(*
SPDX-FileCopyrightText: © 2026 Oleksandr Tiutyk <trofimich@gmail.com>
SPDX-License-Identifier: MIT
License: https://opensource.org/license/mit
*)

FUNCTION_BLOCK StringHelperTest EXTENDS TcUnit.FB_TestSuite
VAR
	{attribute 'hide'} 
	_ClassName : STRING := __POUNAME();
END_VAR

AppendToTarget();
ReplaceInSource();
Split();
Join();
Trim();

METHOD AppendToTarget
VAR
	testString : STRING;

	expectedString : STRING := 'Original string + first appended string + second appended string';
	
	stringToAppend_1 : STRING := 'first appended string';
	stringToAppend_2 : STRING := 'second appended string';
	plusString : STRING := ' + ';
	
	result : BOOL;
END_VAR
VAR_INST
	testFinished : BOOL;
END_VAR
IF testFinished THEN 
	RETURN; 
END_IF 

TEST(__POUNAME());

testString := 'Original string';
TOF_Core.Strings.AppendToTarget255(testString, ' + ', stringToAppend_1, ' + ', stringToAppend_2);
AssertEquals_STRING(expectedString, testString, 'Invalid String.AppendToTarget255 method result');

testString := 'Original string';
result := TOF_Core.Strings.TryAppendToTarget255(testString, ' + ', stringToAppend_1, ' + ', stringToAppend_2);
AssertEquals_STRING(expectedString, testString, 'Invalid String.TryAppendToTarget255 method result');
AssertEquals_BOOL(result, TRUE, 'Invalid String.TryAppendToTarget255 method returned result');

result := TOF_Core.Strings.TryAppendToTarget255(testString, ' + ', stringToAppend_1);
AssertEquals_BOOL(result, FALSE, 'Invalid String.TryAppendToTarget255 method returned result');

testString := 'Original string';
TOF_Core.Strings.AppendToTarget(testString, plusString);
TOF_Core.Strings.AppendToTarget(testString, stringToAppend_1);
TOF_Core.Strings.AppendToTarget(testString, plusString);
TOF_Core.Strings.AppendToTarget(testString, stringToAppend_2);
AssertEquals_STRING(expectedString, testString, 'Invalid String.AppendToTarget method result');

testString := 'Original string';
result := TOF_Core.Strings.TryAppendToTarget(testString, plusString)
	AND TOF_Core.Strings.TryAppendToTarget(testString, stringToAppend_1)
	AND TOF_Core.Strings.TryAppendToTarget(testString, plusString)
	AND TOF_Core.Strings.TryAppendToTarget(testString, stringToAppend_2);
AssertEquals_STRING(expectedString, testString, 'Invalid String.TryAppendToTarget method result');
AssertEquals_BOOL(result, TRUE, 'Invalid String.TryAppendToTarget method returned result');

result := TOF_Core.Strings.TryAppendToTarget(testString, plusString)
	AND TOF_Core.Strings.TryAppendToTarget(testString, stringToAppend_1);
AssertEquals_BOOL(result, FALSE, 'Invalid String.TryAppendToTarget method returned result');

testFinished := TRUE; 
TEST_FINISHED();
END_METHOD

{attribute 'monitoring' := 'call'}
PROPERTY ClassName : REFERENCE TO STRING
GET
ClassName REF= _ClassName;
END_GET
END_PROPERTY

METHOD Join
VAR
	stringToSplit : STRING := '123 , , 456, 789 ,0';
	separator : STRING := ',';
	
	splitter : TOF_Core.StringSplittingEnumerator;

	joinedString1, joinedString2 : STRING;
END_VAR
VAR_INST
	testFinished : BOOL;
END_VAR
IF testFinished THEN 
	RETURN; 
END_IF 

TEST(__POUNAME());

// simple splitting
splitter := TOF_Core.Strings.CreateSplitter(stringToSplit, separator);

// simple joining
TOF_Core.Strings.JoinToTarget(joinedString1, separator, splitter);

AssertEquals_STRING(stringToSplit, joinedString1, TOF_Core.Strings.Concat255('Invalid first Strings.JoinToTarget result string ', joinedString1));

// splitting with maxCount, trimming and empty string removing 
splitter := TOF_Core.Strings.CreateSplitter(stringToSplit, separator, 3, TRUE, TRUE);

// joining with startIndex and count
TOF_Core.Strings.JoinToTarget(joinedString2, separator, splitter, 1, 2);

AssertEquals_STRING('456,789', joinedString2, TOF_Core.Strings.Concat255('Invalid second Strings.JoinToTarget result string ', joinedString2));

testFinished := TRUE;
TEST_FINISHED();
END_METHOD

{attribute 'monitoring' := 'call'}
PROPERTY NamespaceName : REFERENCE TO STRING
GET
NamespaceName REF= CurrentNamespace.Name;
END_GET
END_PROPERTY

METHOD ReplaceInSource
VAR
	testString : STRING(18);
	
	replacementCount : UINT;
	result : BOOL;
END_VAR
VAR_INST
	testFinished : BOOL;
END_VAR
IF testFinished THEN 
	RETURN; 
END_IF 

TEST(__POUNAME());

testString := 'abcd_abcd_abcd';
TOF_Core.Strings.ReplaceInSource(testString, 'bc', '0', replacementCount => replacementCount);
AssertEquals_STRING('a0d_a0d_a0d', testString, 'Invalid String.ReplaceInSource result string');
AssertEquals_UINT(3, replacementCount, 'Invalid String.ReplaceInSource replacingCount count');

testString := 'abcd_abcd_abcd';
TOF_Core.Strings.ReplaceInSource(testString, 'bc', '123', replacementCount => replacementCount);
AssertEquals_STRING('a123d_a123d_a123d', testString, 'Invalid String.ReplaceInSource result string');
AssertEquals_UINT(3, replacementCount, 'Invalid String.ReplaceInSource replacingCount count');

testString := 'abcd_abcd_abcd';
result := TOF_Core.Strings.TryReplaceInSource(testString, 'bc', '0', replacementCount => replacementCount);
AssertEquals_BOOL(TRUE, result, 'Invalid String.TryReplaceInSource result');
AssertEquals_STRING('a0d_a0d_a0d', testString, 'Invalid String.TryReplaceInSource result string');
AssertEquals_UINT(3, replacementCount, 'Invalid String.TryReplaceInSource replacingCount count');

testString := 'abcd_abcd_abcd';
result := TOF_Core.Strings.TryReplaceInSource(testString, 'bc', '123', 1, 1, replacementCount => replacementCount);
AssertEquals_BOOL(TRUE, result, 'Invalid String.TryReplaceInSource result');
AssertEquals_STRING('abcd_a123d_abcd', testString, 'Invalid String.TryReplaceInSource result string');
AssertEquals_UINT(1, replacementCount, 'Invalid String.TryReplaceInSource replacingCount count');

testString := 'abcd_abcd_abcd';
result := TOF_Core.Strings.TryReplaceInSource(testString, 'bc', '1234', replacementCount => replacementCount);
AssertEquals_BOOL(FALSE, result, 'Invalid String.TryReplaceInSource memory handling');

testFinished := TRUE; 
TEST_FINISHED();
END_METHOD

METHOD Split
VAR
	stringToSplit : STRING := '123 , , 456, 789 ,0';
	separator : STRING := ',';
	
	splitter : TOF_Core.StringSplittingEnumerator;
	currentEntry : STRING;
	i : BYTE;
END_VAR
VAR_INST
	testFinished : BOOL;
END_VAR
IF testFinished THEN 
	RETURN; 
END_IF 

TEST(__POUNAME());

// simple splitting
splitter := TOF_Core.Strings.CreateSplitter(stringToSplit, separator);

i := 0;

WHILE splitter.MoveNext() DO
	currentEntry := splitter.CurrentEntry;
	
	CASE i OF
		0:
			AssertEquals_STRING('123 ', currentEntry, 'Invalid StringSplitter entry #0');			
		1:
			AssertEquals_STRING(' ', currentEntry, 'Invalid StringSplitter entry #3');
		2:
			AssertEquals_STRING(' 456', currentEntry, 'Invalid StringSplitter entry #1');
		3:
			AssertEquals_STRING(' 789 ', currentEntry, 'Invalid StringSplitter entry #2');
		4:
			AssertEquals_STRING('0', currentEntry, 'Invalid StringSplitter entry #4');
	END_CASE	
	
	i := i + 1;
END_WHILE

// splitting with maxCount, trimming and empty string removing 
splitter := TOF_Core.Strings.CreateSplitter(stringToSplit, separator, 3, TRUE, TRUE);

i := 0;

WHILE splitter.MoveNext() DO
	currentEntry := splitter.CurrentEntry;
	
	CASE i OF
		0:
			AssertEquals_STRING('123', currentEntry, 'Invalid StringSplitter entry #0');			
		1:
			AssertEquals_STRING('456', currentEntry, 'Invalid StringSplitter entry #1');
		2:
			AssertEquals_STRING('789', currentEntry, 'Invalid StringSplitter entry #2');
		ELSE
			AssertFalse(i > 3, 'Invalid StringSplitter MaxCount handling');
	END_CASE	
	
	i := i + 1;
END_WHILE

testFinished := TRUE;
TEST_FINISHED();
END_METHOD

METHOD Trim
VAR
	trimString : STRING;
END_VAR
VAR_INST
	testFinished : BOOL;
END_VAR
IF testFinished THEN 
	RETURN; 
END_IF 

TEST(__POUNAME());

trimString := '  123   ';
TOF_Core.Strings.TrimChar(trimString, trimMode := TOF_Core.TRIM_MODE.LEFT_AND_RIGHT);
AssertEquals_STRING('123', trimString, 'Invalid string trimming result (TRIM_MODE = LEFT_AND_RIGHT)');			

trimString := '  123   ';
TOF_Core.Strings.TrimChar(trimString, trimMode := TOF_Core.TRIM_MODE.LEFT);
AssertEquals_STRING('123   ', trimString, 'Invalid string trimming result (TRIM_MODE = LEFT)');			

trimString := '  123   ';
TOF_Core.Strings.TrimChar(trimString, trimMode := TOF_Core.TRIM_MODE.RIGHT);
AssertEquals_STRING('  123', trimString, 'Invalid string trimming result (TRIM_MODE = RIGHT)');			

testFinished := TRUE; 
TEST_FINISHED();
END_METHOD

END_FUNCTION_BLOCK

(* stored: Version 1.1.0.1, ProductVersion 3.1.4026.20
   POU StringHelperTest: Id {c2b9cac4-73fd-4d3d-8df7-b5beb6b26c4c}, SpecialFunc None
   Method AppendToTarget: Id {dfc63422-169c-4318-97d7-f4972908ec69}
   Property ClassName: Id {b8985102-dc15-41e1-ae23-7d62e6866a91}
   Get Get: Id {03ded19b-ca6c-4934-9ab2-2e75c95c0490}
   Method Join: Id {ad5df54c-ebe3-4f2b-b686-f2235cc5e4f3}
   Property NamespaceName: Id {02163062-dd40-4429-a0a8-5c360f5da8fb}
   Get Get: Id {459ad87f-22cb-4069-bbe1-8915f5177a12}
   Method ReplaceInSource: Id {acab7dc3-475e-41e3-9ac6-f109a2619017}
   Method Split: Id {afcb1a60-4677-4461-950d-5644dc25733b}
   Method Trim: Id {4efc06d8-47aa-41ec-86fa-bcfd7ab44822} *)
